// TwinCAT 3 PLC project Untitled1
// ProgramVersion: 3.1.4023.0
// libraries:
//   High level object TwinCAT 3 library, * (Tomas Rompotl)
//   Tc2_Standard, * (Beckhoff Automation GmbH)
//   Tc2_System, * (Beckhoff Automation GmbH)
//   Tc3_Module, * (Beckhoff Automation GmbH)
// project tree:
//   / PlcTask.TcTTO
//   POUs/ ListOfTest.TcPOU, MAIN.TcPOU, NodeOfTest.TcPOU
// real-time tasks:
//   TASK PlcTask: cycle T#10ms, priority 20, ADS port 350

CONFIGURATION Untitled1
    RESOURCE PLC ON TwinCAT3
        TASK PlcTask(INTERVAL := T#10ms, PRIORITY := 20);
        PROGRAM MAIN WITH PlcTask : MAIN;
    END_RESOURCE
END_CONFIGURATION

// ---- POUs/MAIN.TcPOU
PROGRAM MAIN
VAR
	testList : List;
	testList2 : ListOfTest;
	
	test : BOOL;
	tesst : TestStructure;
	testinfo : __SYSTEM.VAR_INFO;
	newuser : POINTER TO BYTE;
	
	infoTest : BOOL;
	info : __SYSTEM.VAR_INFO;
	var1 : REAL := 3.14;
	var2 : REAL := 0;
	pInfo : POINTER TO BYTE;
	{attribute 'displaymode':='hex'}
	offset : ULINT;
	pReal : POINTER TO BYTE;
END_VAR

IF test THEN
	test := FALSE;
	testList2.Append(5);
	newuser := __NEW(BYTE, 5);
END_IF



info := __VARINFO(var1);
offset := info.ByteAddress;// + info.ByteOffset;
pInfo := offset;
//MEMCPY(ADR(var2), pInfo, 4); //this works
IF infoTest THEN
	infoTest := FALSE;
	IF info.TypeName = 'REAL' THEN
		pReal := __NEW(REAL);
		MEMCPY(pReal, pInfo, 4); //this not
		var2 := pReal^;
	END_IF
END_IF

END_PROGRAM

// ---- POUs/ListOfTest.TcPOU
FUNCTION_BLOCK ListOfTest EXTENDS List
VAR_INPUT
END_VAR
VAR_OUTPUT
END_VAR
VAR
END_VAR

END_FUNCTION_BLOCK

// ---- POUs/NodeOfTest.TcPOU
FUNCTION_BLOCK NodeOfTest EXTENDS Node
VAR_INPUT
END_VAR
VAR_OUTPUT
END_VAR
VAR
END_VAR

{attribute 'monitoring:= 'variable'}
PROPERTY data : STRING
GET
END_GET
SET
END_SET
END_PROPERTY

END_FUNCTION_BLOCK
